(* Schneider Machine Expert - Basic project Esteira, file version 3.0.0.0 *)
(* ProjectInformations: Name=Esteira de um CD Logistico, Description=Exemplo básico de como funciona um CD logistico, aplicando os conhecimentos de automação. *)
(* UserInformations: LastName=Teodoro, FirstName=Sidney, CellNumber=27996490123, Email=sidneyteodoroaraujojunior2002@gmail.com, City=Belo Horizonte, State=Minags Gerais, Country=Brasil *)

HARDWARE
  Cpu 0: TM221CE16R
  EthernetConfiguration: NetworkName=M221, IpAllocationMode=FixedAddress, IpAddress=0.0.0.0, SubnetMask=0.0.0.0
  SerialLineConfiguration: Baud=Baud19200, Parity=ParityEven, DataBits=DataBits8, StopBits=StopBits1, PhysicalMedium=PhysicalMediumRs485, TransmissionMode=TransmissionModeModbusRtu, SlaveId=1, Addressing=SlaveAddressing
  MastTask: UsePeriodScanMode=false, PeriodScan=100
  FastTask: Period=255
  CpuBehavior: StartingMode=StartAsPreviousState, AutoSaveRamOnEeprom=true, WatchdogPeriod=250

SYMBOLS  (address, symbol, comment, settings)
  %M10      SENSOR1
  %M12      ON_OFF
  %M13      STOP
  %M14      STOP2
  %M15      ON_OFF2
  %M20      MOTOR1
  %M21      MOTOR2
  %M22      MOTOR3
  %M23      MOTOR4
  %M24      MOTOR5
  %M25      MOTOR6
  %M26      MOTOR7
  %M27      MOTOR8
  %M28      MOTOR9
  %M29      MOTOR10
  %TM0        [Preset=3, Base=OneSecond]
  %TM1        [Preset=6, Base=OneSecond]
  %TM2        [Preset=9, Base=OneSecond]
  %TM3        [Preset=12, Base=OneSecond]
  %TM4        [Preset=15, Base=OneSecond]
  %TM5        [Preset=18, Base=OneSecond]
  %TM6        [Preset=21, Base=OneSecond]
  %TM7        [Preset=24, Base=OneSecond]
  %TM8        [Preset=27, Base=OneSecond]
  %TM9        [Preset=30, Base=OneSecond]

POU Novo POU
  (* SectionNumber=1 *)

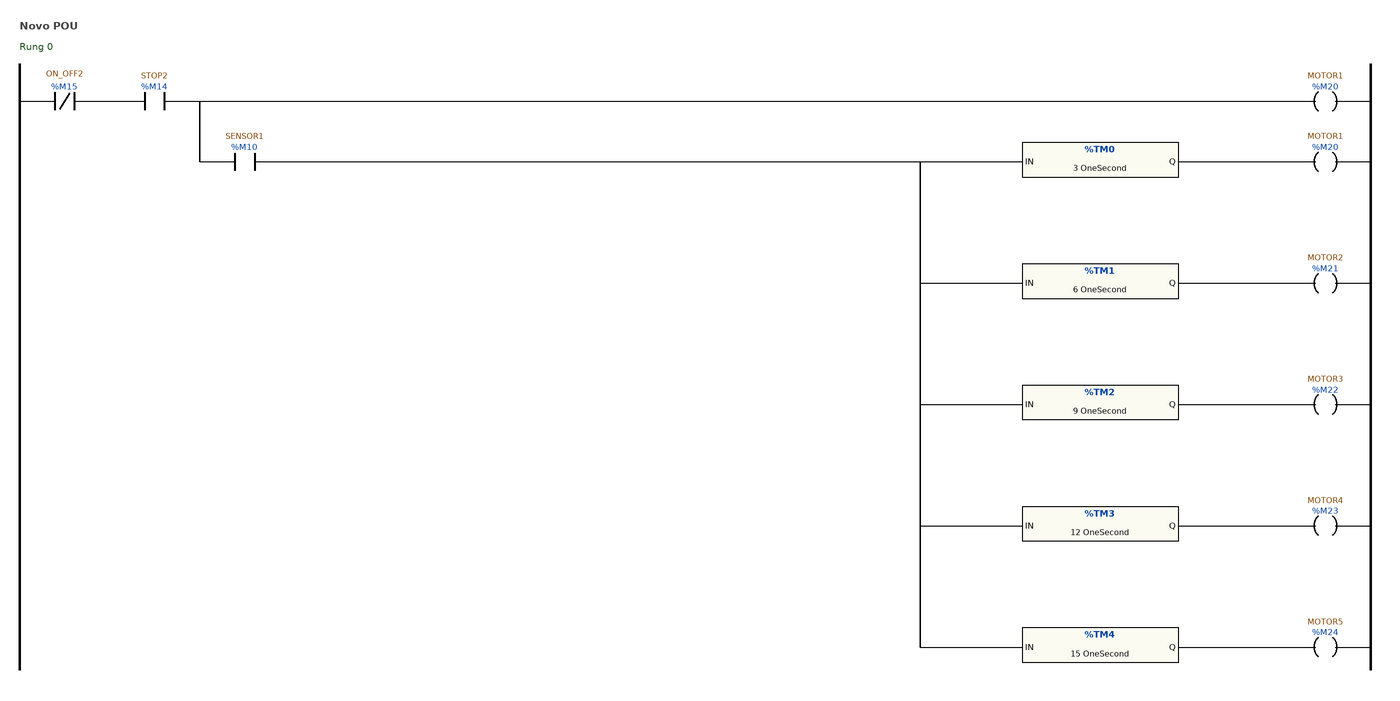

// Rung 0
  LD 1
  MULTIFB
  LD 1
  ANDN %M15               (* ON_OFF2 *)
  AND %M14                (* STOP2 *)
  ST %MW2009:X0
  LD %MW2009:X0
  ST %M20                 (* MOTOR1 *)
  LD %MW2009:X0
  AND %M10                (* SENSOR1 *)
  ST %MW2009:X1
  BLK %TM0
  LD %MW2009:X1
  IN
  OUT_BLK
  LD Q
  ST %M20                 (* MOTOR1 *)
  END_BLK
  BLK %TM1
  LD %MW2009:X1
  IN
  OUT_BLK
  LD Q
  ST %M21                 (* MOTOR2 *)
  END_BLK
  BLK %TM2
  LD %MW2009:X1
  IN
  OUT_BLK
  LD Q
  ST %M22                 (* MOTOR3 *)
  END_BLK
  BLK %TM3
  LD %MW2009:X1
  IN
  OUT_BLK
  LD Q
  ST %M23                 (* MOTOR4 *)
  END_BLK
  BLK %TM4
  LD %MW2009:X1
  IN
  OUT_BLK
  LD Q
  ST %M24                 (* MOTOR5 *)
  END_BLK
  MULTIFB
  // as ST:
  //   MOTOR1 := NOT ON_OFF2 AND STOP2;
  //   %TM0(IN := NOT ON_OFF2 AND STOP2 AND SENSOR1);
  //   MOTOR1 := %TM0.Q;
  //   %TM1(IN := NOT ON_OFF2 AND STOP2 AND SENSOR1);
  //   MOTOR2 := %TM1.Q;
  //   %TM2(IN := NOT ON_OFF2 AND STOP2 AND SENSOR1);
  //   MOTOR3 := %TM2.Q;
  //   %TM3(IN := NOT ON_OFF2 AND STOP2 AND SENSOR1);
  //   MOTOR4 := %TM3.Q;
  //   %TM4(IN := NOT ON_OFF2 AND STOP2 AND SENSOR1);
  //   MOTOR5 := %TM4.Q;

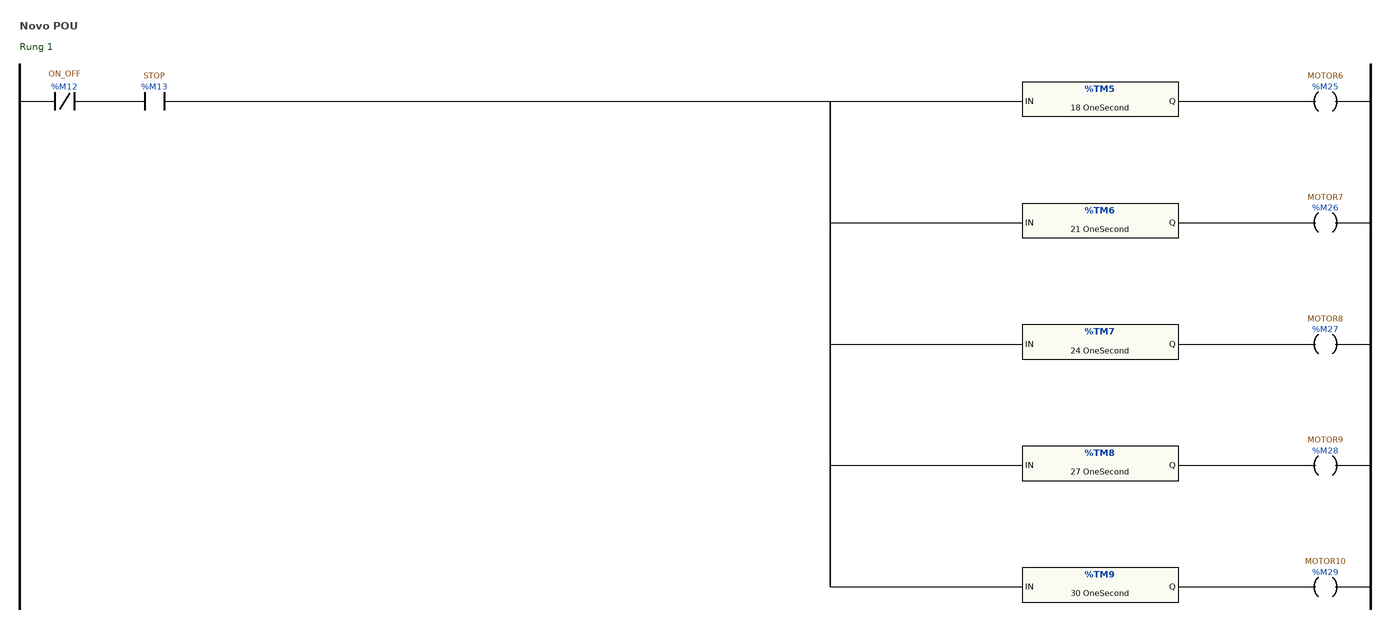

// Rung 1
  LD 1
  MULTIFB
  LD 1
  ANDN %M12               (* ON_OFF *)
  AND %M13                (* STOP *)
  ST %MW2009:X0
  BLK %TM5
  LD %MW2009:X0
  IN
  OUT_BLK
  LD Q
  ST %M25                 (* MOTOR6 *)
  END_BLK
  BLK %TM6
  LD %MW2009:X0
  IN
  OUT_BLK
  LD Q
  ST %M26                 (* MOTOR7 *)
  END_BLK
  BLK %TM7
  LD %MW2009:X0
  IN
  OUT_BLK
  LD Q
  ST %M27                 (* MOTOR8 *)
  END_BLK
  BLK %TM8
  LD %MW2009:X0
  IN
  OUT_BLK
  LD Q
  ST %M28                 (* MOTOR9 *)
  END_BLK
  BLK %TM9
  LD %MW2009:X0
  IN
  OUT_BLK
  LD Q
  ST %M29                 (* MOTOR10 *)
  END_BLK
  MULTIFB
  // as ST:
  //   %TM5(IN := NOT ON_OFF AND STOP);
  //   MOTOR6 := %TM5.Q;
  //   %TM6(IN := NOT ON_OFF AND STOP);
  //   MOTOR7 := %TM6.Q;
  //   %TM7(IN := NOT ON_OFF AND STOP);
  //   MOTOR8 := %TM7.Q;
  //   %TM8(IN := NOT ON_OFF AND STOP);
  //   MOTOR9 := %TM8.Q;
  //   %TM9(IN := NOT ON_OFF AND STOP);
  //   MOTOR10 := %TM9.Q;
